(* PLC project Senza_nome, Sconosciuto Senza_nome 1 *)
(* stored: creationDateTime 2021-03-29T13:33:15, modificationDateTime 2021-03-29T14:46:01 *)

FUNCTION_BLOCK mySquare
  VAR_INPUT
    enable : BOOL;  (* Abilita la generazione di un'onda quadra in uscita *)
  END_VAR
  VAR_OUTPUT
    square : BOOL;  (* Onda quadra in uscita *)
  END_VAR
  VAR
    timeUp : TIME := T#1s;  (* Tempo per cui la variabile square rimane alta *)
    timeDwn : TIME := T#2s;  (* Tempo per cui la variabile square rimane bassa *)
    TON0 : TON;
    TON1 : TON;
  END_VAR

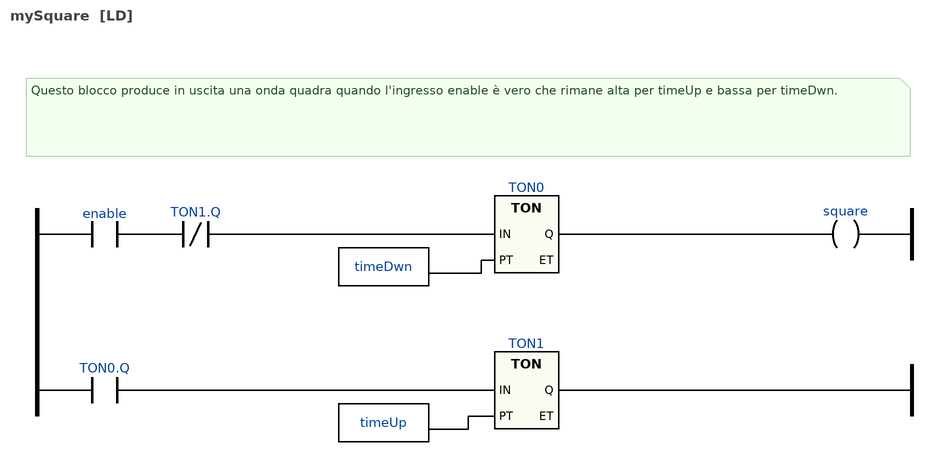
(* LD diagram, written out as Structured Text *)
(* Questo blocco produce in uscita una onda quadra quando l'ingresso enable è vero che rimane alta per timeUp e bassa per timeDwn. *)
TON0(IN := enable AND NOT TON1.Q, PT := timeDwn);
square := TON0.Q;
TON1(IN := TON0.Q, PT := timeUp);
END_FUNCTION_BLOCK

(* Questa funzione implementa lo XOR logico *)
FUNCTION myXOR : BOOL
  VAR_INPUT
    a : BOOL;  (* Primo ingresso della funzione XOR *)
    b : BOOL;  (* Secondo ingresso della funzione XOR *)
  END_VAR

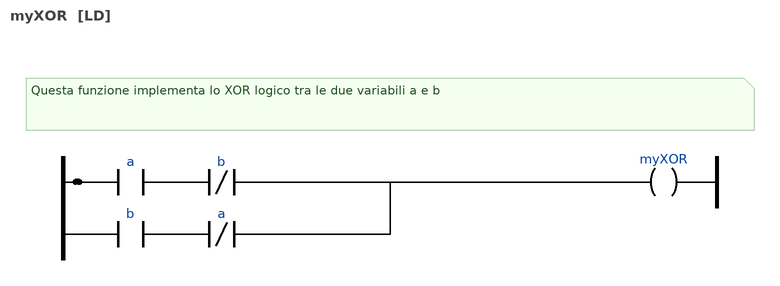
(* LD diagram, written out as Structured Text *)
(* Questa funzione implementa lo XOR logico tra le due variabili a e b *)
myXOR := a AND NOT b OR b AND NOT a;
END_FUNCTION

PROGRAM main
  VAR
    a : BOOL;
    b : BOOL;
    square : BOOL := 0;
    resetCnt : BOOL := 0;
    CNT : INT := 0;
    mySquare0 : mySquare;
    CTU0 : CTU;
  END_VAR
  VAR  (* added by the conversion: wires and edge detectors of the diagram *)
    R_TRIG1 : R_TRIG;
  END_VAR

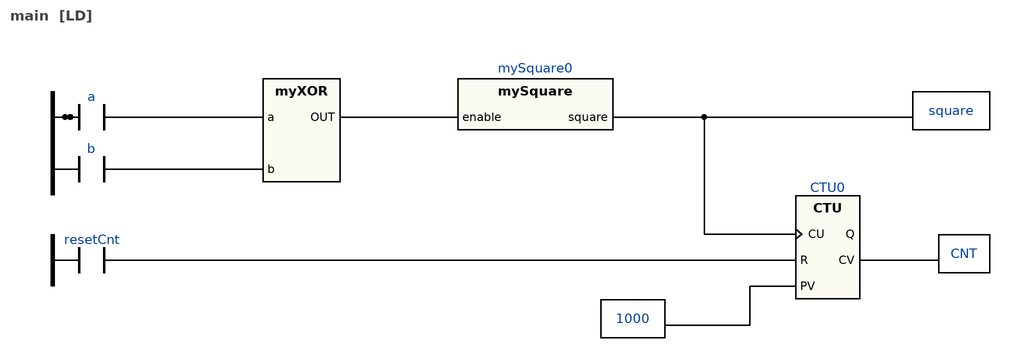
(* LD diagram, written out as Structured Text *)
mySquare0(enable := myXOR(a, b));
square := mySquare0.square;
R_TRIG1(CLK := mySquare0.square);
CTU0(CU := R_TRIG1.Q, R := resetCnt, PV := 1000);
CNT := CTU0.CV;
END_PROGRAM

PROGRAM myST_PRG
  VAR
    a : BOOL;
    b : BOOL;
    enbl : BOOL;
    out : BOOL;
    mySQ : mySquare;
  END_VAR

            (*Chiamata a funzione*)
enbl := myXOR(a := a, 
              b := b);
              
(*Chiamata a blocco funzionale*)
mySQ(enable := enbl, 
     square => out);
          
END_PROGRAM

CONFIGURATION Config0
  RESOURCE Res0 ON PLC
    TASK myTask(INTERVAL := T#20ms, PRIORITY := 0);
    PROGRAM myMainPRGInstance WITH myTask : main;
    PROGRAM mySTPRGInstance WITH myTask : myST_PRG;
  END_RESOURCE
END_CONFIGURATION
